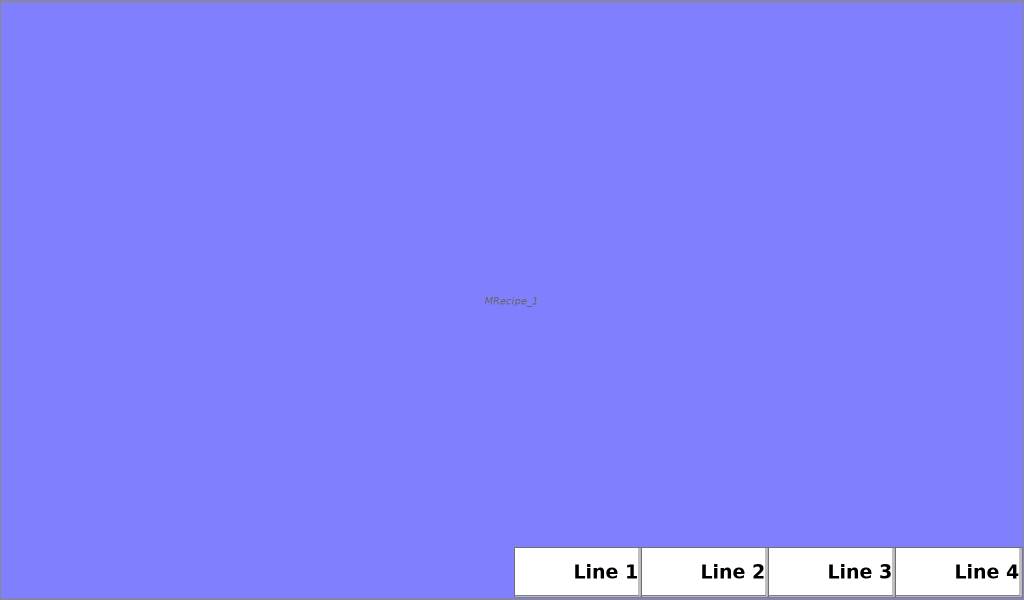
VISUALIZATION MRecipe  // 1024x600
    Frame (0,2 1023x598)
        shows MRecipe_1()
        shows MRecipe_2()
        shows MRecipe_3()
        shows MRecipe_4()
    Button (514,547 127x50), "Line 1", image: VisuSymbols.Symbols.Box
        OnMouseDown: FrameSelectionChange Selection=SelectedFrame=146e207b-fd78-4676-ba16-384fa245d7d2, GlobSel=AssignDir=MainPage.GenElemInst_1003, AssignType=Directly, SelType=Locally
    Button (641,547 127x50), "Line 2", image: VisuSymbols.Symbols.Box
        OnMouseDown: FrameSelectionChange Selection=SelectedFrame=146e207b-fd78-4676-ba16-384fa245d7d2, Selection=1, GlobSel=AssignDir=MainPage.GenElemInst_1003, AssignType=Directly, SelType=Locally
    Button (768,547 127x50), "Line 3", image: VisuSymbols.Symbols.Box
        OnMouseDown: FrameSelectionChange Selection=SelectedFrame=146e207b-fd78-4676-ba16-384fa245d7d2, Selection=2, GlobSel=AssignDir=MainPage.GenElemInst_1003, AssignType=Directly, SelType=Locally
    Button (895,547 127x50), "Line 4", image: VisuSymbols.Symbols.Box
        OnMouseDown: FrameSelectionChange Selection=SelectedFrame=146e207b-fd78-4676-ba16-384fa245d7d2, Selection=3, GlobSel=AssignDir=MainPage.GenElemInst_1003, AssignType=Directly, SelType=Locally
END_VISUALIZATION

(* stored: Version 1.1.0.1, ProductVersion 3.1.4024.12
   Visu MRecipe: Id {59bcd4b8-437b-46a5-a8c2-d3c641f482e1} *)
